{attribute 'qualified_only'}
{attribute 'strict'}
{attribute 'to_string'}
TYPE E_SystemState :
(
    // --- Boot / idle ---------------------------------------------------
    InitController      := 0, 	// Controller Initialization (one-shot config, params, PID setup)
    SesOff              := 70,  // SES Off (idle / standby, waiting for SES ON command)

    // --- Startup sequence ----------------------------------------------
    CheckIfHot          := 10,  // Check if system was just running (hot restart shortcut)
    FillWater       	:= 20,  // SES Initialization - Fill Water
    PurgeVessel     	:= 30,  // SES Initialization - Purge Vessel
    SetDiffPressure 	:= 40,  // SES Initialization - Setting Differential Pressure
    SteamPrecheck       := 50,  // SES Initialization - Main (final checks before flow)

    // --- Run -------------------------------------------------------------
    SteamFlowing        := 60,  // Steam Flowing (normal production, PID flow control)

    // --- Service / abnormal ----------------------------------------------
    Maintenance         := 80,  // Maintenance mode (manual actuation, loopback)
    Fault               := 99   // Fault (latched; operator reset returns to InitController)
	
) INT;
END_TYPE

(* stored: Version 1.1.0.1, ProductVersion 3.1.4026.18
   DUT E_SystemState: Id {6d3cbdae-193b-4d46-b0cc-2b77a8d0c420} *)
